FUNCTION_BLOCK INTERNAL FINAL FB_WriteRepeatedFieldBoolTests EXTENDS FB_TestSuite
VAR_INPUT
END_VAR
VAR_OUTPUT
END_VAR
VAR
	aActual             : ARRAY [0..15] OF BOOL;
    fbFieldCodec 		: FB_FieldCodecBool(nTag:= 16#0A);
	fbRepeatedField		: FB_RepeatedField(anyArray:= F_ToAnyType(aActual), anyFirstElem:= F_ToAnyType(aActual[0]), ipFieldCodec:= fbFieldCodec);
END_VAR

ShouldWriteRepeatedFieldTheory();

METHOD PRIVATE Reset
VAR_INPUT
END_VAR
fbRepeatedField.Initialize();
MEMSET(destAddr:= ADR(aActual), fillByte:= 16#0, n:= SIZEOF(aActual));
END_METHOD

METHOD PRIVATE ShouldWriteRepeatedField
VAR_IN_OUT CONSTANT
    aExpected   : ARRAY [*] OF BYTE;
END_VAR
VAR_INPUT
	aValues     : ARRAY [0..15] OF BOOL;
    nLength     : UDINT;
    nTag        : UDINT;
    nBufferPosStart     : UDINT;
    nExpectedBufferPos  : UDINT;
    ipFieldCodec        : I_FieldCodec;
END_VAR
VAR_INST
    fbCtx   : FB_WriteContext;
END_VAR
VAR
    aActualBuffer       : ARRAY [0..15] OF BYTE;
    hr                  : HRESULT;
END_VAR
// Arrange
Reset();
fbCtx.FromBuffer(aActualBuffer);
fbCtx.refCtx.stState.nBufferPos := nBufferPosStart;
fbRepeatedField.InitializeFromArray(anyArray:= F_ToAnyType(aValues), anyFirstElem:= F_ToAnyType(aValues[0]), nCount:= nLength);
// Act
hr := fbRepeatedField.WriteTo(fbWriteCtx:= fbCtx, ipFieldCodec:= ipFieldCodec);

// Assert
AssertEquals_DINT(
    Expected:= S_OK,
    Actual:= hr,
    Message:= 'Expected S_OK instead of error');
    
{warning disable C0041}
AssertArrayEquals_BYTE(Expecteds:= aExpected, Actuals:= aActualBuffer, Message:= '');
 
AssertEquals_UDINT(
    Expected:= nExpectedBufferPos,
    Actual:= fbCtx.refCtx.stState.nBufferPos,
    Message:= CONCAT('Expected stState.nBufferPos to equal ', TO_STRING(nExpectedBufferPos)));
END_METHOD

METHOD PRIVATE ShouldWriteRepeatedFieldTheory : REFERENCE TO FB_Test
VAR CONSTANT
    cExpectedZeroLength		: ARRAY[0..15] OF BYTE := [16#00, 16#00];
    cExpected1        		: ARRAY[0..15] OF BYTE := [16#00, 16#0A, 16#05, 16#01, 16#00, 16#01, 16#01, 16#00];
END_VAR

VAR CONSTANT
    aZeroLength    			: ARRAY [0..15] OF BOOL := [0, 0, 0, 0, 0, 0, 0, 0, 0, 0, 0, 0, 0, 0, 0, 0];
    aValue1              	: ARRAY [0..15] OF BOOL := [TRUE, FALSE, TRUE, TRUE, FALSE];
END_VAR
TEST(__POUNAME());

ShouldWriteRepeatedField(aExpected:= cExpectedZeroLength, aValues:= aZeroLength, nLength:= 0, nTag:= 1, nBufferPosStart:= 0, nExpectedBufferPos:= 0, ipFieldCodec:= THIS^.fbFieldCodec);
ShouldWriteRepeatedField(aExpected:= cExpected1, aValues:= aValue1, nLength:= 5, nTag:= 1, nBufferPosStart:= 1, nExpectedBufferPos:= 8, ipFieldCodec:= THIS^.fbFieldCodec);

TEST_FINISHED_NAMED(__POUNAME());
END_METHOD

END_FUNCTION_BLOCK

(* stored: Version 1.1.0.1
   POU FB_WriteRepeatedFieldBoolTests: Id {6978f9d6-982f-4766-946e-b9360a2872fd}, SpecialFunc None
   Method Reset: Id {383b7417-471d-48f2-8ed4-752b696a559b}
   Method ShouldWriteRepeatedField: Id {b870bee8-f6ad-4d61-94de-a3b32ba9ea35}
   Method ShouldWriteRepeatedFieldTheory: Id {e090e55e-5430-4bb1-9605-6c7b1b150142} *)
